{attribute 'qualified_only'}
{attribute 'strict'}
TYPE E_PTC_TX_ID :
(
	MAIN_FSM := 16#190,
	Reset := 16#1AB
	
)UINT;
END_TYPE

(* stored: Version 1.1.0.1
   DUT E_PTC_TX_ID: Id {4d7c4aac-d1df-4c3f-9743-e2e23c7beca3} *)
